ABB RobotStudio station: zaliczenie_zadanie1_20200111-160128.rsstn

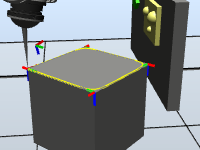
Station zaliczenie_zadanie1 (saved by RobotStudio 6.8.8307.1040)
Controller IRB_6640_185kg_2.80m
  mechanical unit ROB_1: IRB6640_185_280__04, 6 joints, base frame (0, 0, 0) mm
Layout (positions relative to the parent item):
  - IRB6640_185_280__04 [mechanism, from Robots\IRB6640_185_280_G_04.rslib] at (0, 0, 0) mm; joint values [0.7751, 0.0252, 0.7726, -0.3673, 0.8047, 1.8208] (rad or m)
  - Part_13 [part]
  - Part_14 [part] at (132.45, 1287.69, 0) mm
  - Part_20 [part] at (0, 0, 10) mm
  - Part_21 [part] at (0, 0, 10) mm
  - Part_34 [part]
  - dupsko_bonczura [mechanism] at (1081.44, 986.88, 804.35) mm, rotated rx -180 ry 15 rz 135 deg
      TCP dupsko_bonczura at (65.7, 0, 297.48) mm, rotated rx 0 ry 15 rz 0 deg
      links: Part_42
  - Part_48 [part]
  - Part_58 [part]
  - Part_59 [part] at (391.01, 977.32, 0) mm
  - Part_60 [part] at (1091.01, 977.32, 0) mm, rotated rx 0 ry 0 rz 45 deg
Attachment: dupsko_bonczura is attached to IRB6640_185_280__04 / Link6
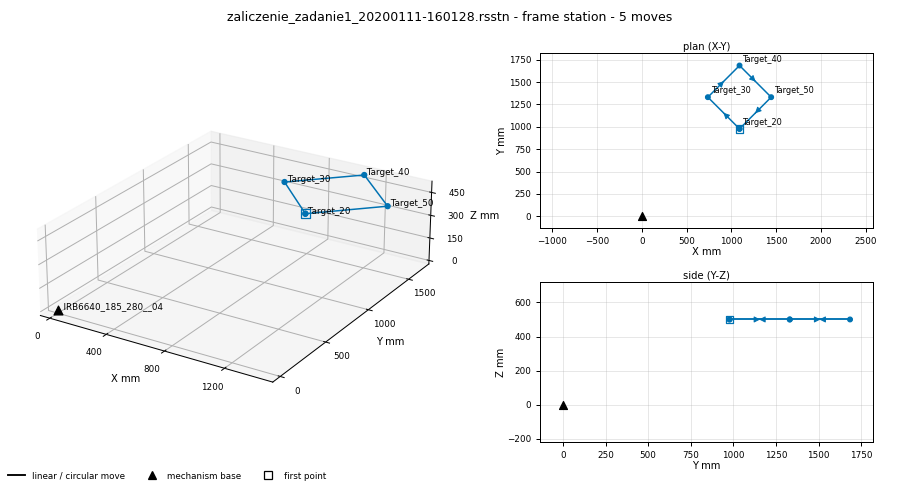
[picture p0: tool path of zaliczenie_zadanie1_20200111-160128.rsstn in frame station, 5 of 5 moves have a stored position in this frame; points joined in program order, loops and branches not executed]
Targets, tools, work objects and paths stored in the station, written as RAPID:
! task T_ROB1
MODULE CalibData
  PERS tooldata MyNewTool:=[TRUE,[[489.305,-400.511,237.057],[0.965925826,0,0.258819045,0]],[1,[0,0,1],[1,0,0,0],0,0,0]];
  PERS tooldata dupsko_bonczura:=[TRUE,[[65.705,0,297.481],[0.991444861,0,0.130526192,0]],[1,[0,0,1],[1,0,0,0],0,0,0]];
ENDMODULE

! task T_ROB1
MODULE Module1
  CONST robtarget Target_10:=[[851.118345102,1020.171978166,1407.621892407],[0.030067918,-0.678210356,0.729882488,-0.079988667],[0,-1,-1,0],[9E+09,9E+09,9E+09,9E+09,9E+09,9E+09]];
  CONST robtarget Target_20:=[[1091.008963611,977.318259815,500],[0,0.382683432,0.923879533,0],[0,0,0,0],[9E+09,9E+09,9E+09,9E+09,9E+09,9E+09]];
  CONST robtarget Target_30:=[[737.455573018,1330.871650409,500],[0,0.382683432,0.923879533,0],[0,0,0,0],[9E+09,9E+09,9E+09,9E+09,9E+09,9E+09]];
  CONST robtarget Target_40:=[[1091.008963611,1684.425041002,500],[0,0.923879533,0.382683432,0],[0,0,0,0],[9E+09,9E+09,9E+09,9E+09,9E+09,9E+09]];
  CONST robtarget Target_50:=[[1444.562354205,1330.871650409,500],[0,0.923879533,-0.382683432,0],[0,0,0,0],[9E+09,9E+09,9E+09,9E+09,9E+09,9E+09]];
  CONST robtarget Target_60:=[[1091.008963611,977.318259815,500],[0,-0.382683432,0.923879533,0],[0,0,0,0],[9E+09,9E+09,9E+09,9E+09,9E+09,9E+09]];
  PROC Path_10()
    MoveL Target_20,v1000,z100,dupsko_bonczura\WObj:=wobj0;
    MoveL Target_30,v1000,z100,dupsko_bonczura\WObj:=wobj0;
    MoveL Target_40,v1000,z100,dupsko_bonczura\WObj:=wobj0;
    MoveL Target_50,v1000,z100,dupsko_bonczura\WObj:=wobj0;
    MoveL Target_60,v1000,z100,dupsko_bonczura\WObj:=wobj0;
  ENDPROC
ENDMODULE

